PROGRAM PISTONS_CYCLE
VAR
	
	bSTARTUP: BOOL:=FALSE;
	counter: INT;
	MANUALcOUNTER:int:=0;
	timimg: REAL:=0.2;
	bTestOpen:BOOL:=TRUE;
	bTestClose:BOOL:=TRUE;
END_VAR

IF NOT bSTARTUP THEN
	
	stPISTON_PARAM[1].nNAME:='FEEDER PUSHER';
	stPISTON_PARAM[1].bOPEN_BY_DEFAULT:=FALSE;
	stPISTON_PARAM[1].openTime:=timimg;
	stPISTON_PARAM[1].closeTime:=timimg;
	stPISTON_PARAM[1].timeoutOpen:=T#3S;
	stPISTON_PARAM[1].timeoutClose:=T#3S;
	stPISTON_PARAM[1].ePISTON_TYPE:= 0;
	
	
	stPISTON_PARAM[2].nNAME:='FEEDER HOLDER';
	stPISTON_PARAM[2].bOPEN_BY_DEFAULT:=FALSE;
	stPISTON_PARAM[2].openTime:=timimg;
	stPISTON_PARAM[2].closeTime:=timimg;
	stPISTON_PARAM[2].timeoutOpen:=T#2S;
	stPISTON_PARAM[2].timeoutClose:=T#2S;
	stPISTON_PARAM[2].ePISTON_TYPE:= 0;
	
	stPISTON_PARAM[15].nNAME:='FEEDER OPENER';
	stPISTON_PARAM[15].bOPEN_BY_DEFAULT:=FALSE;
	stPISTON_PARAM[15].openTime:=timimg;
	stPISTON_PARAM[15].closeTime:=timimg;
	stPISTON_PARAM[15].timeoutOpen:=T#2S;
	stPISTON_PARAM[15].timeoutClose:=T#2S;
	stPISTON_PARAM[15].ePISTON_TYPE:= 0;
	
	stPISTON_PARAM[3].nNAME:='SEPARATE1 LIFT';
	stPISTON_PARAM[3].bOPEN_BY_DEFAULT:=FALSE;
	stPISTON_PARAM[3].openTime:=timimg;
	stPISTON_PARAM[3].closeTime:=timimg;
	stPISTON_PARAM[3].timeoutOpen:=T#3S;
	stPISTON_PARAM[3].timeoutClose:=T#3S;
	stPISTON_PARAM[3].ePISTON_TYPE:= 0;
	
	
	stPISTON_PARAM[4].nNAME:='SEPARATE1 COLET';
	stPISTON_PARAM[4].bOPEN_BY_DEFAULT:=FALSE;
	stPISTON_PARAM[4].openTime:=timimg;
	stPISTON_PARAM[4].closeTime:=timimg;
	stPISTON_PARAM[4].timeoutOpen:=T#3S;
	stPISTON_PARAM[4].timeoutClose:=T#3S;
	stPISTON_PARAM[4].ePISTON_TYPE:= 0;
	
	
	stPISTON_PARAM[5].nNAME:='SEPARATE1 PULL';
	stPISTON_PARAM[5].bOPEN_BY_DEFAULT:=FALSE;
	stPISTON_PARAM[5].openTime:=timimg;
	stPISTON_PARAM[5].closeTime:=timimg;
	stPISTON_PARAM[5].timeoutOpen:=T#3S;
	stPISTON_PARAM[5].timeoutClose:=T#3S;
	stPISTON_PARAM[5].ePISTON_TYPE:= 0;
	
	
	stPISTON_PARAM[6].nNAME:='SEPARATE1 TRAY';
	stPISTON_PARAM[6].bOPEN_BY_DEFAULT:=FALSE;
	stPISTON_PARAM[6].openTime:=timimg;
	stPISTON_PARAM[6].closeTime:=timimg;
	stPISTON_PARAM[6].timeoutOpen:=T#3S;
	stPISTON_PARAM[6].timeoutClose:=T#3S;
	stPISTON_PARAM[6].ePISTON_TYPE:= 0;
	
	
	stPISTON_PARAM[7].nNAME:='SEPARATE1 PUSH PINS';
	stPISTON_PARAM[7].bOPEN_BY_DEFAULT:=FALSE;
	stPISTON_PARAM[7].openTime:=timimg;
	stPISTON_PARAM[7].closeTime:=timimg;
	stPISTON_PARAM[7].timeoutOpen:=T#3S;
	stPISTON_PARAM[7].timeoutClose:=T#3S;
	stPISTON_PARAM[7].ePISTON_TYPE:= 0;
	
	stPISTON_PARAM[16].nNAME:='SEPARATE1 TRAY PUSHER';
	stPISTON_PARAM[16].bOPEN_BY_DEFAULT:=FALSE;
	stPISTON_PARAM[16].openTime:=timimg;
	stPISTON_PARAM[16].closeTime:=timimg;
	stPISTON_PARAM[16].timeoutOpen:=T#3S;
	stPISTON_PARAM[16].timeoutClose:=T#3S;
	stPISTON_PARAM[16].ePISTON_TYPE:= 0;
	
	stPISTON_PARAM[17].nNAME:='SEPARATE1 TRAY DOOR';
	stPISTON_PARAM[17].bOPEN_BY_DEFAULT:=FALSE;
	stPISTON_PARAM[17].openTime:=timimg;
	stPISTON_PARAM[17].closeTime:=timimg;
	stPISTON_PARAM[17].timeoutOpen:=T#3S;
	stPISTON_PARAM[17].timeoutClose:=T#3S;
	stPISTON_PARAM[17].ePISTON_TYPE:= 0;
	
	stPISTON_PARAM[8].nNAME:='SEPARATE2 LIFT';
	stPISTON_PARAM[8].bOPEN_BY_DEFAULT:=FALSE;
	stPISTON_PARAM[8].openTime:=timimg;
	stPISTON_PARAM[8].closeTime:=timimg;
	stPISTON_PARAM[8].timeoutOpen:=T#3S;
	stPISTON_PARAM[8].timeoutClose:=T#3S;
	stPISTON_PARAM[8].ePISTON_TYPE:= 0;
	
	
	stPISTON_PARAM[9].nNAME:='SEPARATE2 COLET';
	stPISTON_PARAM[9].bOPEN_BY_DEFAULT:=FALSE;
	stPISTON_PARAM[9].openTime:=timimg;
	stPISTON_PARAM[9].closeTime:=timimg;
	stPISTON_PARAM[9].timeoutOpen:=T#3S;
	stPISTON_PARAM[9].timeoutClose:=T#3S;
	stPISTON_PARAM[9].ePISTON_TYPE:= 0;
	
	
	stPISTON_PARAM[10].nNAME:='SEPARATE2 PULL';
	stPISTON_PARAM[10].bOPEN_BY_DEFAULT:=FALSE;
	stPISTON_PARAM[10].openTime:=timimg;
	stPISTON_PARAM[10].closeTime:=timimg;
	stPISTON_PARAM[10].timeoutOpen:=T#3S;
	stPISTON_PARAM[10].timeoutClose:=T#3S;
	stPISTON_PARAM[10].ePISTON_TYPE:= 0;
	
	
	stPISTON_PARAM[11].nNAME:='SEPARATE2 TRAY';
	stPISTON_PARAM[11].bOPEN_BY_DEFAULT:=FALSE;
	stPISTON_PARAM[11].openTime:=timimg;
	stPISTON_PARAM[11].closeTime:=timimg;
	stPISTON_PARAM[11].timeoutOpen:=T#3S;
	stPISTON_PARAM[11].timeoutClose:=T#3S;
	stPISTON_PARAM[11].ePISTON_TYPE:= 0;
	
	stPISTON_PARAM[12].nNAME:='SEPARATE2 PUSH PINS';
	stPISTON_PARAM[12].bOPEN_BY_DEFAULT:=FALSE;
	stPISTON_PARAM[12].openTime:=timimg;
	stPISTON_PARAM[12].closeTime:=timimg;
	stPISTON_PARAM[12].timeoutOpen:=T#3S;
	stPISTON_PARAM[12].timeoutClose:=T#3S;
	stPISTON_PARAM[12].ePISTON_TYPE:= 0;
	
	stPISTON_PARAM[18].nNAME:='SEPARATE2 TRAY PUSHER';
	stPISTON_PARAM[18].bOPEN_BY_DEFAULT:=FALSE;
	stPISTON_PARAM[18].openTime:=timimg;
	stPISTON_PARAM[18].closeTime:=timimg;
	stPISTON_PARAM[18].timeoutOpen:=T#3S;
	stPISTON_PARAM[18].timeoutClose:=T#3S;
	stPISTON_PARAM[18].ePISTON_TYPE:= 0;
	
	stPISTON_PARAM[19].nNAME:='SEPARATE2 TRAY DOOR';
	stPISTON_PARAM[19].bOPEN_BY_DEFAULT:=FALSE;
	stPISTON_PARAM[19].openTime:=timimg;
	stPISTON_PARAM[19].closeTime:=timimg;
	stPISTON_PARAM[19].timeoutOpen:=T#3S;
	stPISTON_PARAM[19].timeoutClose:=T#3S;
	stPISTON_PARAM[19].ePISTON_TYPE:= 0;
	
	stPISTON_PARAM[13].nNAME:='DISPOSE OPENER';
	stPISTON_PARAM[13].bOPEN_BY_DEFAULT:=FALSE;
	stPISTON_PARAM[13].openTime:=0.5;
	stPISTON_PARAM[13].closeTime:=0.5;
	stPISTON_PARAM[13].timeoutOpen:=T#3S;
	stPISTON_PARAM[13].timeoutClose:=T#3S;
	stPISTON_PARAM[13].ePISTON_TYPE:= 0;
	
	stPISTON_PARAM[14].nNAME:='CLEAN';
	stPISTON_PARAM[14].bOPEN_BY_DEFAULT:=FALSE;
	stPISTON_PARAM[14].openTime:=timimg;
	stPISTON_PARAM[14].closeTime:=timimg;
	stPISTON_PARAM[14].timeoutOpen:=T#3S;
	stPISTON_PARAM[14].timeoutClose:=T#3S;
	stPISTON_PARAM[14].ePISTON_TYPE:= 0;
	
	stPISTON_PARAM[20].nNAME:='EXTRA ';
	stPISTON_PARAM[20].bOPEN_BY_DEFAULT:=FALSE;
	stPISTON_PARAM[20].openTime:=timimg;
	stPISTON_PARAM[20].closeTime:=timimg;
	stPISTON_PARAM[20].timeoutOpen:=T#3S;
	stPISTON_PARAM[20].timeoutClose:=T#3S;
	stPISTON_PARAM[20].ePISTON_TYPE:= 0;
	
	stPISTON_PARAM[21].nNAME:='DROP PUSHER';
	stPISTON_PARAM[21].bOPEN_BY_DEFAULT:=FALSE;
	stPISTON_PARAM[21].openTime:=0.5;
	stPISTON_PARAM[21].closeTime:=0.5;
	stPISTON_PARAM[21].timeoutOpen:=T#3S;
	stPISTON_PARAM[21].timeoutClose:=T#3S;
	stPISTON_PARAM[21].ePISTON_TYPE:= 0;
	
	stPISTON_PARAM[22].nNAME:='DROP OPENER';
	stPISTON_PARAM[22].bOPEN_BY_DEFAULT:=FALSE;
	stPISTON_PARAM[22].openTime:=timimg;
	stPISTON_PARAM[22].closeTime:=timimg;
	stPISTON_PARAM[22].timeoutOpen:=T#3S;
	stPISTON_PARAM[22].timeoutClose:=T#3S;
	stPISTON_PARAM[22].ePISTON_TYPE:= 0;
	
	FOR counter:=1 TO iNUMBER_OF_PISTONS BY 1 DO
		fbPiston[counter](stPISTON:=stPISTON_PARAM[counter]);
	END_FOR;
	
	bSTARTUP:=TRUE;
END_IF

MANUALcOUNTER:=0;
FOR counter:=1 TO iNUMBER_OF_PISTONS BY 1 DO
	IF fbPiston[counter].bMANUAL THEN
		bManual_mode:=TRUE;
		manualCounter:= manualCounter+1;
	END_IF
	//fbPiston[counter]();
END_FOR;

IF manualCounter = 0 THEN
	bManual_mode:=FALSE;
END_IF
feeder();
clean();
dispose();
feeder();
drop();
separate1();
separate2();

ACTION clean:
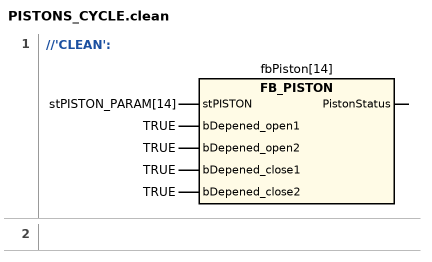
// NETWORK 1
// label: //'CLEAN'
fbPiston[14](
    stPISTON := stPISTON_PARAM[14],
    bDepened_open1 := TRUE,
    bDepened_open2 := TRUE,
    bDepened_close1 := TRUE,
    bDepened_close2 := TRUE); // FB_PISTON

// NETWORK 2
END_ACTION

ACTION dispose:
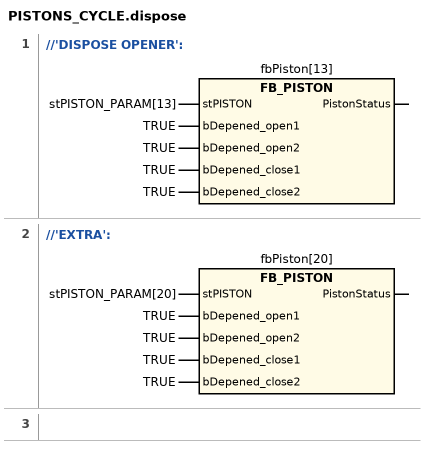
// NETWORK 1
// label: //'DISPOSE OPENER'
fbPiston[13](
    stPISTON := stPISTON_PARAM[13],
    bDepened_open1 := TRUE,
    bDepened_open2 := TRUE,
    bDepened_close1 := TRUE,
    bDepened_close2 := TRUE); // FB_PISTON

// NETWORK 2
// label: //'EXTRA'
fbPiston[20](
    stPISTON := stPISTON_PARAM[20],
    bDepened_open1 := TRUE,
    bDepened_open2 := TRUE,
    bDepened_close1 := TRUE,
    bDepened_close2 := TRUE); // FB_PISTON

// NETWORK 3
END_ACTION

ACTION drop:
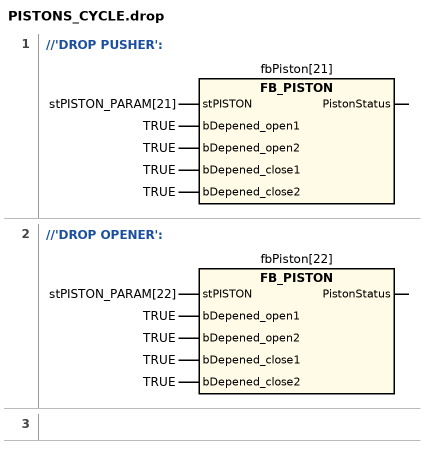
// NETWORK 1
// label: //'DROP PUSHER'
fbPiston[21](
    stPISTON := stPISTON_PARAM[21],
    bDepened_open1 := TRUE,
    bDepened_open2 := TRUE,
    bDepened_close1 := TRUE,
    bDepened_close2 := TRUE); // FB_PISTON

// NETWORK 2
// label: //'DROP OPENER'
fbPiston[22](
    stPISTON := stPISTON_PARAM[22],
    bDepened_open1 := TRUE,
    bDepened_open2 := TRUE,
    bDepened_close1 := TRUE,
    bDepened_close2 := TRUE); // FB_PISTON

// NETWORK 3
END_ACTION

ACTION feeder:
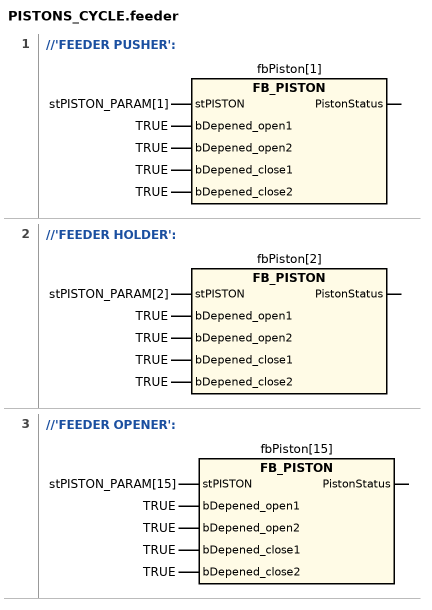
// NETWORK 1
// label: //'FEEDER PUSHER'
fbPiston[1](
    stPISTON := stPISTON_PARAM[1],
    bDepened_open1 := TRUE,
    bDepened_open2 := TRUE,
    bDepened_close1 := TRUE,
    bDepened_close2 := TRUE); // FB_PISTON

// NETWORK 2
// label: //'FEEDER HOLDER'
fbPiston[2](
    stPISTON := stPISTON_PARAM[2],
    bDepened_open1 := TRUE,
    bDepened_open2 := TRUE,
    bDepened_close1 := TRUE,
    bDepened_close2 := TRUE); // FB_PISTON

// NETWORK 3
// label: //'FEEDER OPENER'
fbPiston[15](
    stPISTON := stPISTON_PARAM[15],
    bDepened_open1 := TRUE,
    bDepened_open2 := TRUE,
    bDepened_close1 := TRUE,
    bDepened_close2 := TRUE); // FB_PISTON
END_ACTION

ACTION separate1:
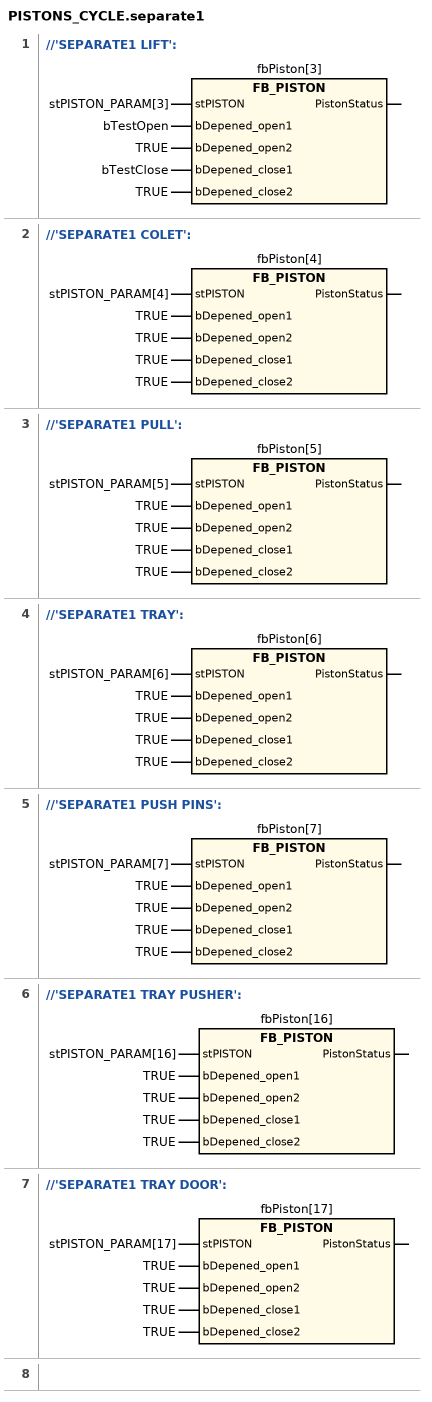
// NETWORK 1
// label: //'SEPARATE1 LIFT'
fbPiston[3](
    stPISTON := stPISTON_PARAM[3],
    bDepened_open1 := bTestOpen,
    bDepened_open2 := TRUE,
    bDepened_close1 := bTestClose,
    bDepened_close2 := TRUE); // FB_PISTON

// NETWORK 2
// label: //'SEPARATE1 COLET'
fbPiston[4](
    stPISTON := stPISTON_PARAM[4],
    bDepened_open1 := TRUE,
    bDepened_open2 := TRUE,
    bDepened_close1 := TRUE,
    bDepened_close2 := TRUE); // FB_PISTON

// NETWORK 3
// label: //'SEPARATE1 PULL'
fbPiston[5](
    stPISTON := stPISTON_PARAM[5],
    bDepened_open1 := TRUE,
    bDepened_open2 := TRUE,
    bDepened_close1 := TRUE,
    bDepened_close2 := TRUE); // FB_PISTON

// NETWORK 4
// label: //'SEPARATE1 TRAY'
fbPiston[6](
    stPISTON := stPISTON_PARAM[6],
    bDepened_open1 := TRUE,
    bDepened_open2 := TRUE,
    bDepened_close1 := TRUE,
    bDepened_close2 := TRUE); // FB_PISTON

// NETWORK 5
// label: //'SEPARATE1 PUSH PINS'
fbPiston[7](
    stPISTON := stPISTON_PARAM[7],
    bDepened_open1 := TRUE,
    bDepened_open2 := TRUE,
    bDepened_close1 := TRUE,
    bDepened_close2 := TRUE); // FB_PISTON

// NETWORK 6
// label: //'SEPARATE1 TRAY PUSHER'
fbPiston[16](
    stPISTON := stPISTON_PARAM[16],
    bDepened_open1 := TRUE,
    bDepened_open2 := TRUE,
    bDepened_close1 := TRUE,
    bDepened_close2 := TRUE); // FB_PISTON

// NETWORK 7
// label: //'SEPARATE1 TRAY DOOR'
fbPiston[17](
    stPISTON := stPISTON_PARAM[17],
    bDepened_open1 := TRUE,
    bDepened_open2 := TRUE,
    bDepened_close1 := TRUE,
    bDepened_close2 := TRUE); // FB_PISTON

// NETWORK 8
END_ACTION

ACTION separate2:
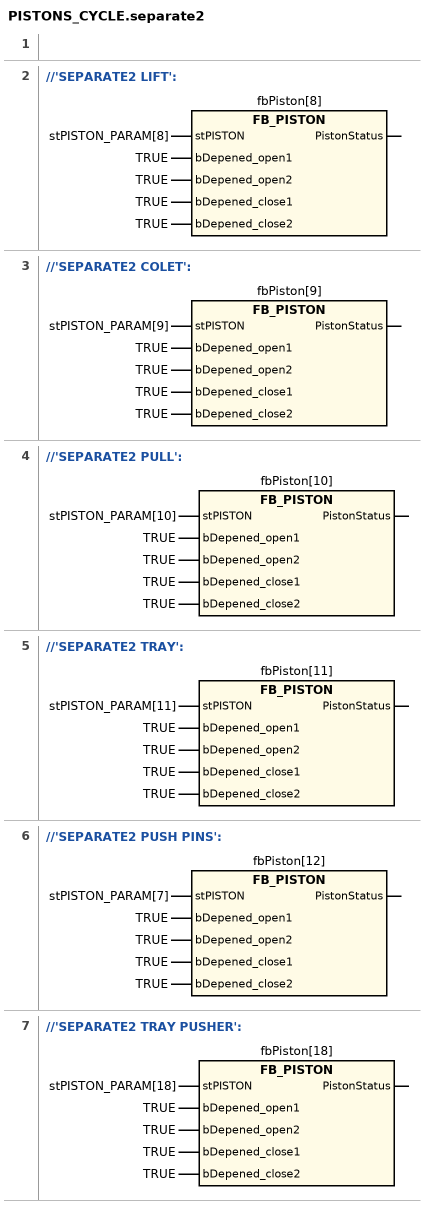
// NETWORK 1

// NETWORK 2
// label: //'SEPARATE2 LIFT'
fbPiston[8](
    stPISTON := stPISTON_PARAM[8],
    bDepened_open1 := TRUE,
    bDepened_open2 := TRUE,
    bDepened_close1 := TRUE,
    bDepened_close2 := TRUE); // FB_PISTON

// NETWORK 3
// label: //'SEPARATE2 COLET'
fbPiston[9](
    stPISTON := stPISTON_PARAM[9],
    bDepened_open1 := TRUE,
    bDepened_open2 := TRUE,
    bDepened_close1 := TRUE,
    bDepened_close2 := TRUE); // FB_PISTON

// NETWORK 4
// label: //'SEPARATE2 PULL'
fbPiston[10](
    stPISTON := stPISTON_PARAM[10],
    bDepened_open1 := TRUE,
    bDepened_open2 := TRUE,
    bDepened_close1 := TRUE,
    bDepened_close2 := TRUE); // FB_PISTON

// NETWORK 5
// label: //'SEPARATE2 TRAY'
fbPiston[11](
    stPISTON := stPISTON_PARAM[11],
    bDepened_open1 := TRUE,
    bDepened_open2 := TRUE,
    bDepened_close1 := TRUE,
    bDepened_close2 := TRUE); // FB_PISTON

// NETWORK 6
// label: //'SEPARATE2 PUSH PINS'
fbPiston[12](
    stPISTON := stPISTON_PARAM[7],
    bDepened_open1 := TRUE,
    bDepened_open2 := TRUE,
    bDepened_close1 := TRUE,
    bDepened_close2 := TRUE); // FB_PISTON

// NETWORK 7
// label: //'SEPARATE2 TRAY PUSHER'
fbPiston[18](
    stPISTON := stPISTON_PARAM[18],
    bDepened_open1 := TRUE,
    bDepened_open2 := TRUE,
    bDepened_close1 := TRUE,
    bDepened_close2 := TRUE); // FB_PISTON

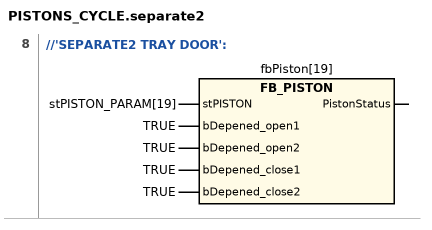
// NETWORK 8
// label: //'SEPARATE2 TRAY DOOR'
fbPiston[19](
    stPISTON := stPISTON_PARAM[19],
    bDepened_open1 := TRUE,
    bDepened_open2 := TRUE,
    bDepened_close1 := TRUE,
    bDepened_close2 := TRUE); // FB_PISTON
END_ACTION

END_PROGRAM

(* stored: Version 1.1.0.1, ProductVersion 3.1.4024.12
   POU PISTONS_CYCLE: Id {b4b09dc6-60ac-43be-9308-062e2f3418e2}, SpecialFunc None
   Action clean: Id {998887aa-8d3b-493b-b070-47ca70dc233d}
   Action dispose: Id {60008ba5-df23-42a5-a8e7-a3896786f315}
   Action drop: Id {8ad63585-fb85-44b7-9ffb-97bf147e413e}
   Action feeder: Id {d7885f46-4b07-41bf-882b-037660cca044}
   Action separate1: Id {afe30f1e-962c-4de7-87ff-61b7ae5ece98}
   Action separate2: Id {b59e5940-8e9f-4bf9-9679-dc5fde737b75} *)
